PROGRAM HMI_1
VAR
END_VAR

// HMI Start 
IF GVL_HMI.NowScreen_NO = 1 THEN 
	GVL_HMI.ChangeScreen_NO := 4 ;
END_IF
// 가이드 축
IF NOT GVL_HMI.AXIS01_LAMP AND NOT GVL_HMI.AXIS02_LAMP AND NOT GVL_HMI.AXIS03_LAMP AND NOT GVL_HMI.AXIS04_LAMP AND NOT GVL_HMI.AXIS05_LAMP THEN
	GVL_HMI.AXIS01_LAMP := 1;
	GVL_HMI.AXIS01 := 1;
END_IF	

IF GVL_HMI.NowScreen_NO = 3030 THEN
	 GVL_HMI.AXIS01_LAMP := 1;
	 GVL_HMI.AXIS02_LAMP := 0;
	 GVL_HMI.AXIS03_LAMP := 0;
	 GVL_HMI.AXIS04_LAMP := 0;
	 GVL_HMI.AXIS05_LAMP := 0;
	 
END_IF

IF GVL_HMI.NowScreen_NO = 3031 THEN
	 GVL_HMI.AXIS01_LAMP := 0;
	 GVL_HMI.AXIS02_LAMP := 1;
	 GVL_HMI.AXIS03_LAMP := 0;
	 GVL_HMI.AXIS04_LAMP := 0;
	 GVL_HMI.AXIS05_LAMP := 0;

END_IF

IF GVL_HMI.NowScreen_NO = 3032 THEN
	 GVL_HMI.AXIS01_LAMP := 0;
	 GVL_HMI.AXIS02_LAMP := 0;
	 GVL_HMI.AXIS03_LAMP := 1;
	 GVL_HMI.AXIS04_LAMP := 0;
	 GVL_HMI.AXIS05_LAMP := 0;

	 
END_IF

IF GVL_HMI.NowScreen_NO = 3033 THEN
	 GVL_HMI.AXIS01_LAMP := 0;
	 GVL_HMI.AXIS02_LAMP := 0;
	 GVL_HMI.AXIS03_LAMP := 0;
	 GVL_HMI.AXIS04_LAMP := 1;
	 GVL_HMI.AXIS05_LAMP := 0;

END_IF

IF GVL_HMI.NowScreen_NO = 3034 THEN
	 GVL_HMI.AXIS01_LAMP := 0;
	 GVL_HMI.AXIS02_LAMP := 0;
	 GVL_HMI.AXIS03_LAMP := 0;
	 GVL_HMI.AXIS04_LAMP := 0;
	 GVL_HMI.AXIS05_LAMP := 1;

END_IF

END_PROGRAM

(* stored: Version 1.1.0.1, ProductVersion 3.1.4024.15
   POU HMI_1: Id {20d5126c-aaf7-4730-921f-2460fcb66fad}, SpecialFunc None *)
